// TIA Portal V19 export
DATA_BLOCK "Area02"   // DB171
// stored: InstanceOfName Area, InstanceOfType FB
"Area"
   // VAR_INPUT
   //    Estop : Bool;
   //    DataIn : Struct
   //       SelMan : Bool;
   //       SelAut : Bool;
   //       PbStart : Bool;
   //       PbStop : Bool;
   //       PbStopProgrammed : Bool;
   //       PbAckRst : Bool;
   //    END_STRUCT;
   //    Config : "AreaConfig";
   //    MachinesStatus : "MachineStatus";
   //    ForceStopInPhase : Bool;
   //    ForceStopProgrammed : Bool;
   //    ResetTimersTimeoutStops : Bool;
   // END_VAR
   // VAR_OUTPUT
   //    AreaInterface { ExternalVisible := 'False'; ExternalWritable := 'False'} : "AreaInterface";
   //    DataOut : Struct
   //       horn : Bool;
   //       lampReady : Bool;
   //       lampCycle : Bool;
   //       LampWarningPresence : Bool;
   //       LampAlarmPresence : Bool;
   //    END_STRUCT;
   //    SilencingAlarms : Bool;
   //    HMI_StatusDinamicText : Int;
   // END_VAR
   // VAR
   //    pbStartOneShotAux : Bool;
   //    RstAlrOneShot1 : Bool;
   //    RstAlrOneShot2 : Bool;
   //    CycleStopImmediately : Bool;
   //    CycleStopInPhase : Bool;
   //    CycleStarted : Bool;
   //    CycleStopProgrammed : Bool;
   //    CycleOn : Bool;
   //    ManAuxPe : Bool;
   //    ManAuxNe : Bool;
   //    ManPositiveEdge : Bool;
   //    ManNegativeEdge : Bool;
   //    AutAuxPe : Bool;
   //    AutAuxNe : Bool;
   //    AutPositiveEdge : Bool;
   //    AutNegativeEdge : Bool;
   //    AlarmLAuxPe : Bool;
   //    CycleAuxPe : Bool;
   //    ResetAlarmsCmd : Bool;
   //    tonDelayPbStart { S7_SetPoint := 'True'} : IEC_TIMER;
   //    tonDelayRstAck { S7_SetPoint := 'True'} : IEC_TIMER;
   //    tonTimeOutStopPhase { S7_SetPoint := 'True'} : IEC_TIMER;
   //    tonTimeOutStopProgr { S7_SetPoint := 'True'} : IEC_TIMER;
   //    tonTimeOutResetAlr { S7_SetPoint := 'True'} : IEC_TIMER;
   // END_VAR
BEGIN
END_DATA_BLOCK
